// TIA Portal V18 export
DATA_BLOCK "Z axis missing layer detection_DB"   // DB101
VERSION : 0.1
// stored: AutoNumber true, DBAccessibleFromOPCUA true, InstanceOfName Z axis missing layer detection, InstanceOfType FB
"Z axis missing layer detection"
   // VAR_INPUT
   //    Mode : DInt;
   //    PrintStarted : Bool;
   //    PrintPaused : Bool;
   //    PrintEnded : Bool;
   //    Z1AxisPosition : DInt;
   //    Z1FeedStep : DInt;
   //    Z1Relative : Bool;
   //    Z2AxisPosition : DInt;
   //    Z2StepSize : DInt;
   //    Z2Relative : Bool;
   //    AmountOfLayers : DInt;
   //    MotionMargin : DInt;
   //    CompensationStepSize : DInt;
   //    PrintingStepSize : DInt;
   // END_VAR
   // VAR_OUTPUT
   //    Z1PredictedFinalPositionMinus : DInt;
   //    Z1PredictedFinalPosition : DInt;
   //    Z1PredictedFinalPositionPlus : DInt;
   //    Z2PredictedFinalPositionMinus : DInt;
   //    Z2PredictedFinalPosition : DInt;
   //    Z2PredictedFinalPositionPlus : DInt;
   //    MissingLayerStatus : Bool;
   //    ErrorTime : Time;
   // END_VAR
   // VAR
   //    CheckSumStart : DInt;
   //    CheckSumMarginPlus : DInt;
   //    CheckSumMarginMinus : DInt;
   //    CheckSumActual : DInt;
   //    MachinePrintingInternal : Bool;
   //    MachinePrintingInternalM1 : Bool;
   //    Z1StartPosition : DInt;
   //    Z2StartPosition : DInt;
   //    Z1AddedDistanceInternal : DInt;
   //    Z2AddedDistanceInternal : DInt;
   // END_VAR
BEGIN
END_DATA_BLOCK
